FUNCTION_BLOCK T_Child
VAR_INPUT
END_VAR
VAR_OUTPUT
END_VAR
VAR

END_VAR

METHOD FB_init : BOOL
VAR_INPUT
    bInitRetains : BOOL; // if TRUE, the retain variables are initialized (warm start / cold start)
    bInCopyCode  : BOOL; // if TRUE, the instance afterwards gets moved into the copy code (online change)
    Counter      : I_Counter;
    Qty          : INT;
END_VAR
Counter.IncCounter(Qty);
END_METHOD

END_FUNCTION_BLOCK

(* stored: Version 1.1.0.1, ProductVersion 3.1.4024.12
   POU T_Child: Id {6df6bf07-349f-4448-9f08-111fc027d888}, SpecialFunc None
   Method FB_init: Id {383e0f0b-8a7c-444e-acd0-ee93468104e7} *)
